# EPICS IOC start-up script: iocsh/ethercatmcOpenClutch.iocsh
ethercatmcCreateAsynParam $(MOTOR_PORT) OpenClutch Int32

dbLoadRecords("ethercatmcOpenClutch.template", "PREFIX=$(PREFIX), AXIS_NAME=$(AXIS_NAME), DESC=$(DESC), MOTOR_PORT=$(MOTOR_PORT), AXIS_NO=$(AXIS_NO)")
